INTERFACE I_GraphicalElement

METHOD PUBLIC RenderTo
VAR_INPUT
	Destination : I_WritableDisplayBuffer;
END_VAR
END_METHOD

METHOD PUBLIC Update
VAR_INPUT
	DeltaTimeInMs : UDINT;
END_VAR
END_METHOD

END_INTERFACE

(* stored: Version 1.1.0.1, ProductVersion 3.1.4024.15
   Itf I_GraphicalElement: Id {503bc0d5-070c-4d9a-aed8-9f6a77673178}
   Method RenderTo: Id {c635a1b8-481b-4dbb-a836-b86a799919c0}
   Method Update: Id {0a6a7d98-db46-444e-bfd6-a1e2a2fc39cc} *)
